PROGRAM P_GantryDiffSup
VAR
	fbXGantryMonitor	:	FB_GantryDifferenceMonitor;
	fbYGantryMonitor	:	FB_GantryDifferenceMonitor;
END_VAR



fbXGantryMonitor(Gantry:=XGantry);
fbYGantryMonitor(Gantry:=YGantry);

END_PROGRAM

(* stored: Version 1.1.0.1, ProductVersion 3.1.4020.12
   POU P_GantryDiffSup: Id {954b9861-204f-4ae9-b8f5-f376391fb77a}, SpecialFunc None *)
